TEXTLIST TextList_Effluvage
  0 = ''
  1 = 'EFFLUVAGE' | FR: 'EFFLUVAGE' | EN: 'GLOW DISCHARGE'
  2 = 'Courant' | FR: 'Courant' | EN: 'Current'
  3 = 'time' | FR: 'Temps' | EN: 'Timer'
  4 = 'PT' | FR: 'Temps écoulé' | EN: 'Passed time'
  5 = 'Tension attendue' | FR: 'Tension attendue' | EN: 'Expected voltage'
  6 = ''
  7 = ''
   = ''
END_TEXTLIST

(* stored: Version 1.1.0.1, ProductVersion 3.1.4024.11
   TextList TextList_Effluvage: Id {de79a1a7-2d2d-4fbb-9779-4b89d333b217} *)
